// TIA Portal V19 export
DATA_BLOCK "CarriageLub_Pump"   // DB130
// stored: InstanceOfName Lubr_Pump, InstanceOfType FB
"Lubr_Pump"
   // VAR_INPUT
   //    DataIn : Struct
   //       SensorLevel : Bool;
   //    END_STRUCT;
   //    ValveCycleTimeOut : Time;
   //    Simulation : Bool;
   // END_VAR
   // VAR_OUTPUT
   //    ValveCmd : Bool;
   // END_VAR
   // VAR_IN_OUT
   //    Par : "LubrPump_Par";
   // END_VAR
   // VAR
   //    Ctrl : Struct
   //       RunReq : Bool;
   //    END_STRUCT;
   //    Sts : Struct
   //       OldValve : Int;
   //    END_STRUCT;
   //    Alarm : "LubrPump_Alr";
   //    HMI : "LubrMotorPump_HMI";
   //    LubrInterface : "LubrValve_ITF";
   //    tonLowLevel : IEC_TIMER;
   //    tonValveON : IEC_TIMER;
   //    tonValveOFF : IEC_TIMER;
   //    ValveChianTimeOut : IEC_TIMER;
   // END_VAR
BEGIN
END_DATA_BLOCK
